# EPICS autosave request: iocBoot/ioc13SXDiff/auto_positions.req
file "CARS_motor_positions.req",         P=$(P), M=m1
~
